TEXTLIST tlPML_States
  0 = 'PMLState_Undefined'
  1 = 'PMLState_Clearing'
  2 = 'PMLState_Stopped'
  3 = 'PMLState_Starting'
  4 = 'PMLState_Idle'
  5 = 'PMLState_Suspended'
  6 = 'PMLState_Execute'
  7 = 'PMLState_Stopping'
  8 = 'PMLState_Aborting'
  9 = 'PMLState_Aborted'
  10 = 'PMLState_Holding'
  11  = 'PMLState_Held'
  12 = 'PMLState_Unholding'
  13 = 'PMLState_Suspending'
  14 = 'PMLState_Unsuspending'
  15 = 'PMLState_Resetting'
  16 = 'PMLState_Completing'
  17 = 'PMLState_Complete'
   = ''
END_TEXTLIST

(* stored: Version 1.1.0.1, ProductVersion 3.1.4024.11
   TextList tlPML_States: Id {76aa32f0-566d-4351-9339-4f179fa22a81} *)
